# EPICS autosave request: keithley2400/k2461_settings.req
$(P):OUTP
$(P):SENS_FUNC
$(P):SENS_PROT
$(P):SENS_RANG
$(P):SENS_RANG_AUTO
$(P):SETX
$(P):SOTX
$(P):SOUR_FUNC
$(P):SOUR_LEV
$(P):SOUR_MODE
$(P):SOUR_RANG
